PROGRAM PRG_HMIControl
VAR
	bHomeBlueLamp	:	BOOL;
END_VAR


IF NOT bHomeBlueLamp THEN
    bHomeBlueLamp := TRUE;
ELSE
    bHomeBlueLamp := FALSE;
END_IF;

GVL_HMIVariables.bHomeLampBlueState := bHomeBlueLamp;

END_PROGRAM

(* stored: Version 1.1.0.1, ProductVersion 3.1.4024.15
   POU PRG_HMIControl: Id {978beb02-d146-472c-ad6b-2f8739fa70ac}, SpecialFunc None *)
